Fanuc KAREL source: kt00408.KL

-- PROVISIONAL review KL for V770-1; original PC SHA256 921bcb8bcb3e506184b34f6bedf5bcbc0f257b27a156a0a86f1ff9aacbfa0113
-- Incomplete behavior may be omitted. Consult companion uncertainty JSON. Do not deploy.
PROGRAM KT00408
%NOLOCKGROUP
VAR
  R1 : REAL
  OUT : BOOLEAN
-- UNRESOLVED_DECL H2 type=002017
BEGIN
  -- UNRESOLVED_PC offsets 5-16; opcodes 2E,23
  -- UNRESOLVED_PC offsets 21-35; opcodes 2E,22,9D,33,B4
  -- UNRESOLVED_PC offsets 40-63; opcodes 21,22,9D,33,B3,64,71,23
  -- UNRESOLVED_PC offsets 68-72; opcodes 7F
END KT00408
